FUNCTION TryConvert_TIME_TO_INT : BOOL
VAR_INPUT
	in : TIME;
	out : REFERENCE TO INT;
END_VAR

IF in > DatatypeLimits.MAX_VALUE_OF_TIME_WHICH_CAN_BE_HELD_IN_A_INT THEN
	RETURN;
END_IF

out := TIME_TO_INT(in);
TryConvert_TIME_TO_INT := TRUE;

END_FUNCTION

(* stored: Version 1.1.0.1, ProductVersion 3.1.4024.12
   POU TryConvert_TIME_TO_INT: Id {d9ee368f-ee36-41ca-9c47-fb8dfc7e23e5}, SpecialFunc None *)
